{attribute 'qualified_only'}
{attribute 'strict'}
TYPE E_Blink :
(
	off := 0,
	slow,
	fast,
	short,
	long,
	on
);
END_TYPE

(* stored: Version 1.1.0.1, ProductVersion 3.1.4024.9
   DUT E_Blink: Id {f099207a-59d9-4c3d-9616-afac1f67bd49} *)
